(* IEC 61131-3 sources: AX2TIA-demo/src, 3 files *)

(* ---- ClassLib.st ---- *)
NAMESPACE ExampleClassLib
    CLASS Belt
       METHOD PUBLIC RunForward ; END_METHOD
       METHOD PUBLIC RunBackward ; END_METHOD
       METHOD PUBLIC Stop ; END_METHOD
    END_CLASS

    CLASS ABSTRACT Conveyor
       METHOD PUBLIC ABSTRACT Run END_METHOD
       METHOD PUBLIC ABSTRACT Stop END_METHOD
    END_CLASS

    CLASS OneBeltConveyor EXTENDS Conveyor
       VAR PUBLIC
          belt : REF_TO Belt;
       END_VAR

       METHOD PUBLIC OVERRIDE Run
         belt^.RunForward();
       END_METHOD

       METHOD PUBLIC OVERRIDE Stop
          belt^.Stop();
       END_METHOD
    END_CLASS

    CLASS TwoBeltConveyor EXTENDS Conveyor
       VAR PUBLIC
          belt1 : REF_TO Belt;
          belt2 : REF_TO Belt;
       END_VAR

       METHOD PUBLIC OVERRIDE Run
          belt1^.RunForward();
          belt2^.RunBackward();
       END_METHOD

       METHOD PUBLIC OVERRIDE Stop
          belt1^.Stop();
          belt2^.Stop();
       END_METHOD
    END_CLASS
 END_NAMESPACE

(* ---- WrapperFB.st ---- *)
NAMESPACE ExampleClassLib.Entry
    FUNCTION_BLOCK EquipmentModule1 // Wrapper FB
       VAR_INPUT
          start : BOOL;
          stop : BOOL;
       END_VAR
       VAR // OK, classes can be instantiated in VAR
          belt1, belt2, belt3 : Belt;
          feed                : OneBeltConveyor;
          transport           : TwoBeltConveyor;
          init                : BOOL := TRUE;
       END_VAR

       IF init THEN
          init := FALSE;
          feed.belt := REF(belt1);
          transport.belt1 := REF(belt2);
          transport.belt2 := REF(belt3);
       END_IF;

       IF start AND NOT stop THEN
          feed.Run();
          // code to move the belt
          transport.Run();
       ELSIF stop THEN
          transport.Stop();
          // code to stop the belt
          feed.Stop();
       END_IF;
    END_FUNCTION_BLOCK
 END_NAMESPACE

(* ---- wrapperFBWithInterface.st ---- *)
USING ExampleClassLib.Entry;
USING ExampleClassLib;
    // Wrapper FB
NAMESPACE ExampleClassLib
    FUNCTION_BLOCK EquipmentModule2 // Wrapper FB
        VAR_INPUT
           start : BOOL;
           stop : BOOL;
        END_VAR
        VAR // OK, interfaces can be declared in VAR
           beltInst : BeltImpl;
           belt     : IBelt1;
           feed     : OneBeltConveyor1;
           init     : BOOL := TRUE;
        END_VAR

        IF init THEN
           init := FALSE;
           belt := beltInst;  // initialize interface
           feed.belt := belt; // use interface
        END_IF;

        IF start AND NOT stop THEN
           feed.Run();
        ELSIF stop THEN
           feed.Stop();
        END_IF;
     END_FUNCTION_BLOCK
END_NAMESPACE
